// TIA Portal V18 export
DATA_BLOCK "FB0-MR_Quantity Control_1_DB"   // DB24
VERSION : 0.1
// stored: AutoNumber true, DBAccessibleFromOPCUA true, InstanceOfName FB0-MR_Quantity Control_1, InstanceOfType FB
"FB0-MR_Quantity Control_1"
   // VAR_INPUT
   //    RatioCheckMode : Int;
   //    AcceptValue : Bool;
   //    "Mixing Ratio 100:B" : Real;
   //    "Qty A set" : Real;
   //    "Qty B set" : Real;
   //    "Pump size A" : Real;
   //    "Pump size B" : Real;
   //    RatioCheckStarted : Bool;
   //    DeleteCalibrationA : Bool;
   //    DeleteCalibrationB : Bool;
   // END_VAR
   // VAR_OUTPUT
   //    "Max. Mixed quantity" : Real;
   //    "Pump Capacity A cc/rev" : Real;
   //    "Pump capacity B cc/rev" : Real;
   //    "cc/rev A" : Real;
   //    "cc/rev B" : Real;
   //    "pump adj. ratio A" : Real;
   //    "pump adj. ratio B" : Real;
   //    "Total Deviation A" : Real;
   //    "Total Deviation B" : Real;
   //    "Current Deviation A" : Real;
   //    "Current Deviation B" : Real;
   //    AllowedMaxAQtyOn2kMetering : Real;
   //    AllowedMaxBQtyOn2kMetering_1 : Real;
   // END_VAR
   // VAR_IN_OUT
   //    "Qty real A" : Real;
   //    "Qty real B" : Real;
   // END_VAR
   // VAR RETAIN
   //    "Last_Cc/rev_A" : Real;
   //    "Last_Cc/rev_B" : Real;
   // END_VAR
   // VAR
   //    "A_Qty/rev_Theor" : Real;
   //    "B_Qty/rev_Theor" : Real;
   //    A_Calc_Ref_rev : Real;
   //    B_Calc_Ref_rev : Real;
   //    A_Total_Deviation : Real;
   //    B_Total_Deviation : Real;
   // END_VAR
   // VAR RETAIN
   //    B_Current_Deviation : Real;
   //    A_Current_Deviation : Real;
   //    "CC/rev actual A" : Real;
   //    "CC/rev actual B" : Real;
   // END_VAR
   // VAR
   //    "A_cc/revStatic_Found" : Real;
   //    "B_cc/revStatic_Found" : Real;
   //    "cc/rev calc A" : Real;
   //    "cc/rev calc B" : Real;
   //    "Maximum capacity Pump A" : Real;
   //    "Maximum capacity Pump B" : Real;
   //    "Individual quantity A MR" : Real;
   //    "Individual quantity B1 MR" : Real;
   //    "Individual quantity B MR" : Real;
   //    "capacity difference" : Real;
   //    "Ratio margin" : Real;
   //    "Ratio/100" : Real;
   //    "Pump cc/rev A" : Real;
   //    "pump cc/rev B" : Real;
   //    "A Quantity Compensated" : Real;
   //    "Quantity A Per ratio" : Real;
   //    Temp_1 : Bool;
   //    Last_DeviationA : Real;
   //    Last_DeviationB : Real;
   // END_VAR
BEGIN
END_DATA_BLOCK
